{attribute 'qualified_only'}
VAR_GLOBAL	
	B1 AT %Q*: BOOL; 	// Füllstand
	B2 AT %Q*: BOOL;    // Position Dose
	S1 AT %Q*: BOOL;    // Taster Reset
	S2 AT %Q*: BOOL;    // Taster Start
END_VAR

(* stored: Version 1.1.0.1, ProductVersion 3.1.4024.5
   GVL DI: Id {c2d05302-d374-4f85-80dd-41006a3e3277} *)
